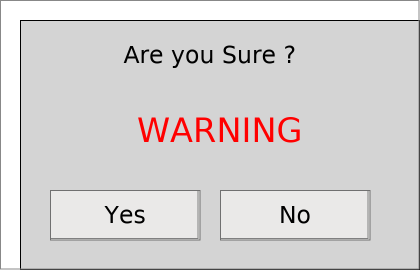
VISUALIZATION CONFIRMATION  // 420x270
VAR_IN_OUT
	result : STRING;
END_VAR
    Rectangle (20,20 400x250)
    Button (50,190 150x50), "Yes"
        toggle OP_BTN.Start_btn
        OnMouseClick: CloseDialog Dialog=CONFIRMATION, Result=Yes, NumpadKeypadSet=True
    Label (85,30 250x50), "Are you Sure ?"
    Button (220,190 150x50), "No"
        OnMouseClick: CloseDialog Dialog=CONFIRMATION, Result=No, NumpadKeypadSet=True
    Textfield (20,100 400x60), "WARNING"
END_VISUALIZATION

(* stored: Version 1.1.0.1, ProductVersion 3.1.4024.12
   Visu CONFIRMATION: Id {97e414c8-b6af-4fb5-a504-2dd77bcb83b1} *)
